TYPE ST_MC_ParametersAxis :
STRUCT
	
	

END_STRUCT
END_TYPE

(* stored: Version 1.1.0.1, ProductVersion 3.1.4024.12
   DUT ST_MC_ParametersAxis: Id {1dd533a3-f30c-45d0-b9f6-087478b2a3a3} *)
